(* IEC 61131-3 sources: CodigoPPC/Variaveis, 8 files *)

(* ---- GVL_Alarm.st ---- *)
{attribute 'qualified_only'}
VAR_GLOBAL
    // ─────────────────────────────────────────────────────────
    // ALARM MANAGER FLAGS (condições booleanas)
    // ─────────────────────────────────────────────────────────

	// Falhas na inicialização
    WARN_INV_CHECK_PARTIAL          : BOOL := FALSE;  // Inversores ausentes mas acima do limiar
	CRIT_SERIAL_INIT_FAIL			: BOOL := FALSE;	// Critico - Falha para iniciar as seriais
	CRIT_K1_TIMEOUT 				: BOOL := FALSE;    // Critico - falha na inicialização de K1 - falta detectar fechamento
	CRIT_K2_TIMEOUT 				: BOOL := FALSE;    // Critico - falha na inicialização de K2 - falta detectar fechamento
    CRIT_INV_CHECK_BELOW_THRESHOLD  : BOOL := FALSE;  // Respondentes < limiar → stError

    // Medição / Medidor
    ALARM_MEAS_MODBUS_TIMEOUT      	: BOOL := FALSE;  	// timeout de leitura (READ)
    ALARM_MEAS_MODBUS_ERRO       	: BOOL := FALSE;  	// xError do medidor (READ)
    ALARM_MEAS_FROZEN	            : BOOL := FALSE;  	// diagnosticCode = A900 (se aplicável)
    ALARM_MEAS_USING_LAST_VALUEU	: BOOL := FALSE;  	// bPoucosErros=TRUE e bDadosOK=FALSE
	ALARM_MEAS_RANGE_ERROR    		: BOOL := FALSE;    // Warning: Valor fora de faixa
    ALARM_MEAS_XCHECK_FAIL   		: BOOL := FALSE;    // Warning: Validação cruzada
    CRIT_MEAS_PERSISTENT_FAIL		: BOOL := FALSE;  	// bPoucosErros = FALSE
    CRIT_MEAS_MODBUS_TIMEOUT      	: BOOL := FALSE;  	// timeout de leitura (READ) repeticao fora da tolerancia
    CRIT_MEAS_MODBUS_ERRO       	: BOOL := FALSE;  	// xError do medidor (READ)  repeticao fora da tolerancia
	CRIT_MEAS_INIC_ERRO_TIMEOUT		: BOOL := FALSE;    // falha no teste de comunicação na inicialização do medidor

    // Comunicação inversores
    CRIT_COM_CHANNEL_FAIL           : BOOL := FALSE;  	// falha geral de comunicação → FAIL/STOP
	CRIT_CH1_MODBUS_TIMEOUT        	: BOOL := FALSE; 	// Canal COM1 TIMEOUT 3x
    CRIT_CH2_MODBUS_TIMEOUT        	: BOOL := FALSE; 	// Canal COM2 TIMEOUT 3x
	CRIT_CH1_MODBUS_ERRO	       	: BOOL := FALSE;  	// >50% falhas COM1 no ciclo
    CRIT_CH2_MODBUS_ERRO        	: BOOL := FALSE;  	// >50% falhas COM2 no ciclo

    // Sistema
	ALARM_SCAN_OVERRUN        		: BOOL := FALSE;    // Warning: Watchdog de ciclo
    CRIT_TC_POWER_NOT_SET           : BOOL := FALSE;    // TC_Power_kW = 0 na inicialização
    CRIT_NO_INVERTERS        		: BOOL := FALSE;    // Error: Nenhum inversor configurado
    CRIT_RTC_FAIL            		: BOOL := FALSE;    // Error: Falha RTC
    CRIT_INSTALLED_PWR_ZERO  		: BOOL := FALSE;    // Error: Potência instalada = 0
	CRIT_INSTALLED_SMAX_ZERO  		: BOOL := FALSE;    // Error: Potência reativa instalada = 0
	CRIT_SCAN_OVERRUN        		: BOOL := FALSE;    // CRITICO: Watchdog de ciclo 3x

    // Proteções normativas
    CRIT_HARDLIMIT_15S       		: BOOL := FALSE;    // Error: P > LPI+10% por >15s
    CRIT_EXPORT_OVER_LPI_30S   		: BOOL := FALSE;    // Error: P > LPI por >30s
    CRIT_K2_NOT_OPENED       		: BOOL := FALSE;    // Error: K2 não abriu após trip
	CRIT_MEAS_TIMEOUT_IN_FAIL    	: BOOL := FALSE;	// 5s sem medição válida em FAIL → STOP
	CRIT_FAIL_ENTRY                 : BOOL := FALSE;    // Entrada no estado FAIL

	// Status do sistema
	ALARM_FAIL_ACTIVE				: BOOL := FALSE;  	// MachineState=FAIL
    CRIT_STOP_ACTIVE	            : BOOL := FALSE;  	// MachineState=STOP
	CRIT_SCHEDULE_INDEX_INVALID		: BOOL := FALSE;    // Dia ou hora da semana inválido (CRITICAL)

    // ── Controle / PF ──
    ALARM_PF_BELOW_TARGET     		: BOOL := FALSE;    // Warning: PF < 0.92
    ALARM_PF_CRITICAL         		: BOOL := FALSE;    // Error: PF < 0.92 + Q saturado
    ALARM_Q_LIMITED_BY_SMAX    		: BOOL := FALSE;    // Info: Q limitado por S

	// FAIL-SAFE avançado
	ALARM_FAIL_RECOVERY_STARTED     : BOOL := FALSE;    // Timer de recuperação iniciou
	CRIT_FAIL_WRITE_FAILED          : BOOL := FALSE;    // Escrita zero falhou (inversores não responderam)
	CRIT_FAIL_WRITE_EXHAUSTED       : BOOL := FALSE;    // Esgotou retentativas de escrita zero → STOP
	CRIT_FAIL_GLOBAL_TIMEOUT        : BOOL := FALSE;    // Permaneceu em FAIL além do máximo permitido

	    // ── TURNOFF ──
    ALARM_TURNOFF_ACTIVE            : BOOL := FALSE;    // MachineState = TURNOFF
    CRIT_TURNOFF_WRITE_EXHAUSTED    : BOOL := FALSE;    // Escrita zero esgotou tentativas
    CRIT_TURNOFF_VERIFY_TIMEOUT     : BOOL := FALSE;    // Timeout verificação geração
    CRIT_TURNOFF_K2_NOT_OPENED      : BOOL := FALSE;    // K2 não abriu após trip controlado
	CRIT_TURNOFF_K1_NOT_OPENED      : BOOL := FALSE;    // K1 não abriu após comando

END_VAR

(* ---- GVL_ALARM_MANAGER.st ---- *)
{attribute 'qualified_only'}
VAR_GLOBAL
    // ─────────────────────────────────────────────────────────
    // ALARM MANAGER FLAGS (condições booleanas)
    // ─────────────────────────────────────────────────────────

	// Falhas na inicialização
	CRIT_SERIAL_INIT_FAIL			: BOOL := FALSE;	// Critico - Falha para iniciar as seriais
	CRIT_K1_TIMEOUT 				: BOOL := FALSE;    // Critico - falha na inicialização de K1 - falta detectar fechamento
	CRIT_K2_TIMEOUT 				: BOOL := FALSE;    // Critico - falha na inicialização de K2 - falta detectar fechamento

    // Medição / Medidor
    ALARM_MEAS_MODBUS_TIMEOUT      	: BOOL := FALSE;  	// timeout de leitura (READ)
    ALARM_MEAS_MODBUS_ERRO       	: BOOL := FALSE;  	// xError do medidor (READ)
    ALARM_MEAS_FROZEN	            : BOOL := FALSE;  	// diagnosticCode = A900 (se aplicável)
    ALARM_MEAS_USING_LAST_VALUEU	: BOOL := FALSE;  	// bPoucosErros=TRUE e bDadosOK=FALSE
	ALARM_MEAS_RANGE_ERROR    		: BOOL := FALSE;    // Warning: Valor fora de faixa
    ALARM_MEAS_XCHECK_FAIL   		: BOOL := FALSE;    // Warning: Validação cruzada
    CRIT_MEAS_PERSISTENT_FAIL		: BOOL := FALSE;  	// bPoucosErros = FALSE
    CRIT_MEAS_MODBUS_TIMEOUT      	: BOOL := FALSE;  	// timeout de leitura (READ) repeticao fora da tolerancia
    CRIT_MEAS_MODBUS_ERRO       	: BOOL := FALSE;  	// xError do medidor (READ)  repeticao fora da tolerancia

    // Comunicação inversores
    CRIT_COM_CHANNEL_FAIL           : BOOL := FALSE;  	// falha geral de comunicação → FAIL/STOP
	CRIT_CH1_MODBUS_TIMEOUT        	: BOOL := FALSE; 	// Canal COM1 TIMEOUT 3x
    CRIT_CH2_MODBUS_TIMEOUT        	: BOOL := FALSE; 	// Canal COM2 TIMEOUT 3x
	CRIT_CH1_MODBUS_ERRO	       	: BOOL := FALSE;  	// >50% falhas COM1 no ciclo
    CRIT_CH2_MODBUS_ERRO        	: BOOL := FALSE;  	// >50% falhas COM2 no ciclo

    // Sistema
	ALARM_SCAN_OVERRUN        		: BOOL := FALSE;    // Warning: Watchdog de ciclo
    CRIT_TC_POWER_NOT_SET           : BOOL := FALSE;    // TC_Power_kW = 0 na inicialização
    CRIT_NO_INVERTERS        		: BOOL := FALSE;    // Error: Nenhum inversor configurado
    CRIT_RTC_FAIL            		: BOOL := FALSE;    // Error: Falha RTC
    CRIT_INSTALLED_PWR_ZERO  		: BOOL := FALSE;    // Error: Potência instalada = 0
	CRIT_INSTALLED_SMAX_ZERO  		: BOOL := FALSE;    // Error: Potência reativa instalada = 0
	CRIT_SCAN_OVERRUN        		: BOOL := FALSE;    // CRITICO: Watchdog de ciclo 3x

    // Proteções normativas
    CRIT_HARDLIMIT_15S       		: BOOL := FALSE;    // Error: P > LPI+10% por >15s
    CRIT_EXPORT_OVER_LPI_30S   		: BOOL := FALSE;    // Error: P > LPI por >30s
    CRIT_K2_NOT_OPENED       		: BOOL := FALSE;    // Error: K2 não abriu após trip
	CRIT_MEAS_TIMEOUT_IN_FAIL    	: BOOL := FALSE;	// 5s sem medição válida em FAIL → STOP
	CRIT_FAIL_ENTRY                 : BOOL := FALSE;    // Entrada no estado FAIL

	// Status do sistema
	ALARM_FAIL_ACTIVE				: BOOL := FALSE;  	// MachineState=FAIL
    CRIT_STOP_ACTIVE	            : BOOL := FALSE;  	// MachineState=STOP
	CRIT_SCHEDULE_INDEX_INVALID		: BOOL := FALSE;    // Dia ou hora da semana inválido (CRITICAL)

    // ── Controle / PF ──
    ALARM_PF_BELOW_TARGET     		: BOOL := FALSE;    // Warning: PF < 0.92
    ALARM_PF_CRITICAL         		: BOOL := FALSE;    // Error: PF < 0.92 + Q saturado
    ALARM_Q_LIMITED_BY_SMAX    		: BOOL := FALSE;    // Info: Q limitado por S
END_VAR

(* ---- GVL_Comm.st ---- *)
{attribute 'qualified_only'}
(* ═══════════════════════════════════════════════════════════════════════
   GVL_Comm — Área de dados da comunicação Modbus RTU programática
   ═══════════════════════════════════════════════════════════════════════
   Esta GVL é o ponto de interface entre a Task_ModbusComm (que executa
   a comunicação) e a Task_Main (que executa o controle).

   Capacidade:
   COM1: 1 medidor + até 15 inversores
   COM2: até 15 inversores
   Canais de escrita por inversor: até 20 (índices 0..19)

   REGRA DE CONCORRÊNCIA (escritor único):
     - Task_ModbusComm ESCREVE: bCOMxConnected, bMeterOnline,
       bMeterReadDone, eMeterResult, awMeterRawData,
       bInvReadDone_COMx, eInvResult_COMx
     - Task_Main ESCREVE: bWritePendingCOMx, setpoints
     - Task_ModbusComm LÊ: bWritePendingCOMx, setpoints
   ═══════════════════════════════════════════════════════════════════════ *)
{attribute 'qualified_only'}

VAR_GLOBAL CONSTANT
    MAX_INV_PER_COM     	: UINT := 15;       // Inversores por porta COM
    MAX_WRITE_CHANNELS  	: UINT := 20;       // Canais de escrita por inversor (0..19)
END_VAR

VAR_GLOBAL
    // ─── Estado das portas COM ───────────────────────────────────
    bCOM1Connected      : BOOL;
    bCOM2Connected      : BOOL;
    bCOM1Error          : BOOL;
    bCOM2Error          : BOOL;

    // ─── Medidor (COM1) — Buffer raw para UN_chint/UN_URP1439 ───
    bMeterOnline        : BOOL;
    bMeterReadDone      : BOOL;
    eMeterResult        : E_ModbusResult;
    awMeterRawData      : ARRAY[0..63] OF WORD;
    uiMeterRegsRead     : UINT;

    // ─── Inversores COM1 — status de resposta ────────────────────
    abInvOnline_COM1        : ARRAY[1..15] OF BOOL;
    uiInvOnlineCount_COM1   : UINT;

    // ─── Inversores COM2 — status de resposta ────────────────────
    abInvOnline_COM2        : ARRAY[1..15] OF BOOL;
    uiInvOnlineCount_COM2   : UINT;

    // ─── Escrita — flags de pendência ────────────────────────────
    bWritePendingCOM1   : BOOL;
    bWritePendingCOM2   : BOOL;

    // ─── Configuração de slaves (preenchidos no stInit) ──────────
    uiMeterSlaveId      : UINT := 100;
    auiInvSlaveIdsCOM1  : ARRAY[1..15] OF UINT;
    auiInvSlaveIdsCOM2  : ARRAY[1..15] OF UINT;
    auiWriteRegAddr     : ARRAY[0..19] OF UINT;    // Endereço de registro por canal (0..19)

    // ─── Configuração geral ──────────────────────────────────────
    bConfigLoaded       : BOOL;
    bCommInitDone       : BOOL;
END_VAR

(* ---- GVL_Log.st ---- *)
{attribute 'qualified_only'}
// ════════════════════════════════════════════════════════════════════
// GVL_EventLog — Constantes do sistema de log de eventos
// ════════════════════════════════════════════════════════════════════
// Autor: Eng. Principal / Revisão Técnica PPC-GD
// Plataforma: WAGO CC100 (751-9402) / CODESYS V3.5 SP21 Patch 4
//
// DIMENSIONAMENTO:
//   64 entradas × 28 bytes = ~1.792 bytes de RETAIN
//   WAGO CC100 possui ~32 kB RETAIN → uso < 6%
//   Com ~1 evento/min, cobre >1 hora de histórico completo
//   Com taxa de pico (~10 eventos em cascata), ainda retém >6 min
// ════════════════════════════════════════════════════════════════════
{attribute 'qualified_only'}
VAR_GLOBAL CONSTANT
    MAX_EVENT_ENTRIES   : UINT := 64;   // Tamanho do ring buffer (potência de 2 facilita debug)
END_VAR

(* ---- GVL_Main.st ---- *)
{attribute 'qualified_only'}
VAR_GLOBAL CONSTANT

    // Parâmetros do sistema
    SOFTVERSION          		: UINT := 21;   					// Versão da aplicação
	DATAAPLICATION				: DATE := DATE#2025-12-05;			// Data da aplicação
	NMAXINVERSORES				: UINT := 30;						// Capacidade máxima de inversores
	TIPOSINVERSORES				: UINT := 8;						// total de inversores diferentes que podem estar presentes
	NDATASESPECIAIS 			: UINT := 48; 						// Quantidade de datas especiais disponíveis ao todo (para 10 anos)
	TIMEZONEOFFSET				: DINT := -3;
    CYCLE_TIME_MS				: UDINT := 1000;  					// tempo de ciclo de controle
	MAX_Meas_MODBUS_ERROS		: UDINT := 3;						// quantidade de erros permitido na leitura do medidor
	MAX_Meas_MODBUS_TIMEOUTS	: UDINT := 3;						// quantidade de timeouts permitido na leitura do medidor

END_VAR

VAR_GLOBAL
	timestampUTC				: UDINT;
	Result 						: RTS_IEC_RESULT;
  	ControlCycle    			: REAL:=1;            					// Tempo de ciclo de controle em SEGUNDOS (ex: 1.0 = 1 segundo)
	MachineState				: E_MachineState:= E_MachineState.START;
	fbEventLog 					: FB_EventLog;						// Function Block de registro de eventos

	CYCLE_TIME_TOLERANCE		: UDINT := 1200;  					// tolerancia de ultrapassagem para tempo de ciclo de controle de 20%

	// Saidas digitais
  	K1_out  					: BOOL;   							// DI X5_1 - K1 - controle permissivo
	K2_out						: BOOL;								// DI X5_2 - K2 - controle trip
  	LedRedOut					: BOOL;								// DI X5_3 - nada pronto - K1 e K2 abertos
  	LedYellowOut  				: BOOL;   							// DI X5_4 - K1 fechou - permissivo ok
  	LedGreenOut  				: BOOL;   							// DI X5_5 - K2 fechou - acende verde -tudo pronto

	// Entredas digitais
	K1_in        				: BOOL;                				// DI X12_1 - contato auxliar de K1_in=1 => K1 fechado (permite gerar)
  	K2_in        				: BOOL;                				// DI X12_2 - contato auxliar de K2_in=1 => K2 fechado (permite gerar) trip desarmado

    // Comandos da IHM
    // ─────────────────────────────────────────────────────────────
  	HMI_StartResetButton     	: BOOL := FALSE;           			// DI X12_3 - botao frontal para comandar ligar/reset geral quando no estado STOP
    HMI_TurnOffButton    		: BOOL := FALSE;  					// DI X12_4 "Desligar controlado"

    //    Medições (REAL) - Tensões (V), Correntes (A), Potências Ativas (W), Potências Reativas (var), PF (adimensional, sinal: + indutivo, - capacitivo)

    Ua  			: REAL := 0.0; // Tensão de fase A   - 2006H - Tensão de fase A em Volts (x 0,1 V)
    Ub  			: REAL := 0.0; // Tensão de fase B   - 2008H - Tensão de fase B em Volts (x 0,1 V)
    Uc  			: REAL := 0.0; // Tensão de fase C   - 200AH - Tensão de fase C em Volts (x 0,1 V)

	Ia    			: REAL 	:= 0.0; // 200CH - Corrente de fase A em A (x 0,001 A)
	Ib    			: REAL 	:= 0.0; // 200EH - Corrente de fase B em A (x 0,001 A)
	Ic    			: REAL 	:= 0.0; // 2010H - Corrente de fase C em A (x 0,001 A)

	Pt    			: REAL 	:= 0.0; // 2012H - Potencia ativa combinada em kW (x 0.1 para W, x 0.0001 para kW)
	Pa    			: REAL 	:= 0.0; // 2014H - Potencia ativa fase A 	em kW (x 0.1 para W, x 0.0001 para kW)
	Pb    			: REAL 	:= 0.0; // 2016H - Potencia ativa fase B 	em kW (x 0.1 para W, x 0.0001 para kW)
	Pc    			: REAL 	:= 0.0; // 2018H - Potencia ativa fase C    em kW (x 0.1 para W, x 0.0001 para kW)

	Qt    			: REAL 	:= 0.0; // 201AH - Potencia reativa combinada em kvar (x 0.1 para var, x 0.0001 para kvar)
	Qa    			: REAL 	:= 0.0; // 201CH - Potencia reativa fase A	 em kvar (x 0.1 para var, x 0.0001 para kvar)
	Qb    			: REAL 	:= 0.0; // 201EH - Potencia reativa fase B	 em kvar (x 0.1 para var, x 0.0001 para kvar)
	Qc    			: REAL 	:= 0.0; // 2020H - Potencia reativa fase C	 em kvar (x 0.1 para var, x 0.0001 para kvar)

	PFt    			: REAL 	:= 0.0; // 202AH - Fator de potência combinado (número positivo: indutivo, número negativo: capacitivo) (x0,001)
	PFa    			: REAL 	:= 0.0; // 202CH - Fator de potência de fase A (número positivo: indutivo, número negativo: capacitivo) (x0,001)
	PFb    			: REAL 	:= 0.0; // 202EH - Fator de potência de fase B (número positivo: indutivo, número negativo: capacitivo) (x0,001)
	PFc    			: REAL 	:= 0.0; // 2030H - Fator de potência de fase C (número positivo: indutivo, número negativo: capacitivo) (x0,001)

	// definição medidores dos dois canais de comunicação
	trigMedidor100  : BOOL;
	pMedidor100		: POINTER TO ModbusSlaveComPort;
	trigMedidor200  : BOOL;
	pMedidor200		: POINTER TO ModbusSlaveComPort;

	// definição dos inversores dos dois canais de comunicação
	MAX_CH1_MODBUS_ERROS		: UINT := 0;						// < 50% da quantidade de inversores sem ir para FAIL
	MAX_CH1_MODBUS_TIMEOUTS		: UINT := 0;						// < 50% da quantidade de inversores sem ir para FAIL
	MAX_CH2_MODBUS_ERROS		: UINT := 0;						// < 50% da quantidade de inversores sem ir para FAIL
	MAX_CH2_MODBUS_TIMEOUTS		: UINT := 0;						// < 50% da quantidade de inversores sem ir para FAIL
	trigInvCOM100				: ARRAY[1..15, 0..4] OF BOOL;
	trigInvCOM200				: ARRAY[1..15, 0..4] OF BOOL;
	NInversoresCOM01    		: UINT :=0;
	NInversoresCOM02    		: UINT :=0;
    pInversores100 	: ARRAY [1..15] OF POINTER TO ModbusSlaveComPort; 				// array de pointers para Inversor01..Inversor15 (apenas ponteiros - não recria instâncias)
	pInversores200 	: ARRAY [1..15] OF POINTER TO ModbusSlaveComPort; 				// array de pointers para Inversor01..Inversor15 (apenas ponteiros - não recria instâncias)

    //   COMANDOS E TELEMETRIA - Saídas do Controle

	// Potencia Total instalada e potencia Aparente Total instalada
  	InstalledPower 	: REAL; 														// Soma da potência nominal de todos os inversores ativos
	Q_max_permitido : REAL := 0.0;    												// Q máximo permitido (kvar)
	InstalledSmax   : REAL; 														// NOVO: Potência Aparente Máxima Total (kVA)

	// COMANDOS DE CONTROLE
	MaxExportLimit 	: REAL;              											// Limite de exportação do scheduler (kW)
	P_cmd_total_kW 	: REAL;              											// Comando total de P (kW)
	Q_cmd_total_kvar: REAL;            												// Comando total de Q (kvar)

    // Telemetria: Setpoint atual da agenda (antes das proteções)
    TotalPowerPercent : REAL;

    // Telemetria: Potência Reativa total desejada (kVA)
    TotalReactivePower : REAL;

    // Telemetria: Valores efetivos calculados para cada inversor
    P_inv_kW     	: ARRAY[1..NMAXINVERSORES] OF REAL; 							// valor de setpoint de potencia ativa em kW
	P_inv_Percent 	: ARRAY[1..NMAXINVERSORES] OF REAL; 							// valor de setpoint de potencia ativa em percentual do nominal
	P_inv_limit 	: ARRAY[1..NMAXINVERSORES] OF REAL; 							// valor limite de potencia ativa com base na SMAX de cada um
    Q_inv_kvar    	: ARRAY[1..NMAXINVERSORES] OF REAL; 							// valor de setpoint de potencia reativa em kVA
    PF_inv 			: ARRAY[1..NMAXINVERSORES] OF REAL; 							// valor do fator de potencia de cada inversor (deve ser 0,92 para todos)
	PF_inv_Percent	: ARRAY[1..NMAXINVERSORES] OF REAL; 							// valor de setpoint de fator de potencia em percentual

	// Margem de segurança para compensar erro de TC perto de zero, o sistema tentará manter importação mínima garantido que não haja exportação
	SafetyMargin_pct: REAL :=0.03;
	TC_Power_kW		: REAL := 0.0; // deve ser configurado como 3% da potencia total sob controle pelo TC

	// ════════════════════════════════════════════════════════════════
	// DIAGNÓSTICO DE PF
	// ════════════════════════════════════════════════════════════════
	Q_available_max : REAL;             											// Q máximo disponível (kvar)
	PF_effective 	: REAL;                											// PF efetivo resultante
	PFErro 			: BOOL;                   										// TRUE = PF < 0.92 não atingível (banco de capacitores)

	// ════════════════════════════════════════════════════════════════
    // DIAGNÓSTICO DE FATOR DE POTÊNCIA
    // ════════════════════════════════════════════════════════════════

    // Status geral
    PF_target : REAL := 0.92;                   // PF alvo (mínimo aceitável)
    PF_measured : REAL;                         // PF medido no ponto de conexão
    PF_achieved : REAL;                         // PF efetivamente alcançado após compensação
    PF_OK : BOOL;                               // TRUE = PF ≥ 0.92

    // Potências
    P_generated_kW : REAL;                      // P total gerado pelos inversores
    P_allocated_kW : REAL;                      // P efetivamente alocado
    Q_measured_kvar : REAL;                     // Q medido no ponto de conexão (carga)
    Q_required_kvar : REAL;                     // Q necessário para atingir PF ≥ 0.92
    Q_commanded_kvar : REAL;                    // Q comandado pelo FB_PIQ
    Q_available_kvar : REAL;                    // Q que inversores conseguem fornecer
    Q_allocated_kvar : REAL;                    // Q efetivamente alocado
    Q_deficit_kvar : REAL;                      // Déficit de Q (se > 0, falta Q)

    // Capacidade dos inversores
    S_total_available_kVA : REAL;               // S total disponível (soma de todos inversores)
    S_total_used_kVA : REAL;                    // S total utilizado
    S_utilization_pct : REAL;                   // % de utilização de S
    Q_capacity_total_kvar : REAL;               // Capacidade total de Q dos inversores (atual)
    Q_utilization_pct : REAL;                   // % de utilização de Q

    // Diagnóstico e recomendações
    Q_deficit_percent : REAL;                   // Déficit de Q em % do necessário
    Capacitor_bank_size_kvar : REAL;            // Tamanho recomendado de banco de capacitores
    Capacitor_bank_recommended : BOOL;          // TRUE = Recomenda banco de capacitores
    PF_alarm_code : UINT;                       // Código de alarme (0=OK, 1=Aviso, 2=Crítico)

    // Histórico (opcional)
    PF_min_24h : REAL := 1.0;                   // PF mínimo nas últimas 24h
    PF_avg_24h : REAL := 1.0;                   // PF médio nas últimas 24h
    Q_deficit_max_24h : REAL;                   // Déficit máximo de Q nas últimas 24h
    PF_alarm_count_24h : UDINT;                 // Quantidade de alarmes nas últimas 24h

    // Inversores individuais (diagnóstico detalhado)
    Inv_S_utilization : ARRAY[1..NMAXINVERSORES] OF REAL;  // % S usado por inversor
    Inv_Q_available : ARRAY[1..NMAXINVERSORES] OF REAL;    // Q disponível por inversor (kvar)
    Inv_limited : ARRAY[1..NMAXINVERSORES] OF BOOL;        // TRUE = Inversor limitado por S
END_VAR

(* ---- GVL_ModbusProfiles.st ---- *)
(* ═══════════════════════════════════════════════════════════════════════
   GVL_ModbusProfiles — Perfis de dispositivos Modbus
   ═══════════════════════════════════════════════════════════════════════
   Contém os perfis hardcoded de cada modelo de inversor suportado.
   Declarados como CONSTANT: imutáveis em runtime, residem em Flash.

   FASE 1: apenas Goodwe GW50K-MT (único modelo em operação).
   FASE 4: FB_LoadProfiles substituirá estes valores por dados do CSV,
           mantendo este como fallback em caso de falha de leitura.

   PROTOCOLO GOODWE — REGISTRO 0x0101 (Fator de Potência):
     Indutivo  (Q ≥ 0): valor 80..100 → PF = valor / 100  (ex: 92 → PF 0.92)
     Capacitivo(Q < 0): valor  1.. 20 → PF = (100-valor)/100 (ex: 10 → PF 0.90 cap)
     A conversão para este formato já é feita pelo FB_QAlloc e armazenada
     em GVL_Main.PF_inv_Percent[i]. Aqui Scale=1.0 pois o valor já está
     no formato correto para o registro.

   PROTOCOLO GOODWE — REGISTRO 0x0100 (Potência Ativa):
     Valor direto 0..100 representando 0..100% da potência nominal.
     FB_PAlloc já calcula P_inv_Percent em 0..100. Scale=1.0.
   ═══════════════════════════════════════════════════════════════════════ *)
{attribute 'qualified_only'}
VAR_GLOBAL CONSTANT

    Profile_Goodwe_GW50K : ST_InverterProfile := (
        Name             := 'Goodwe GW50K-MT',
        ManufacturerCode := 1,          // 1 = Goodwe
        MaxRegsPerWrite  := 1,          // Goodwe: 1 registro por transação FC06
        InterFrameDelayMs := 0,         // ModbusFB respeita silêncio RTU automaticamente

        nWriteRegs := 2,
        WriteMap := [
            // Índice 0 — Setpoint Potência Ativa (%)
            (Address     := 16#0100,    // 256 decimal
             Quantity    := 1,
             FuncCode    := 6,          // FC06: Write Single Register
             Scale       := 1.0,        // P_inv_Percent já está em 0..100
             Offset      := 0.0,
             MinPhys     := 0.0,        // 0% = inversor parado
             MaxPhys     := 100.0,      // 100% = potência nominal
             bEnabled    := TRUE),

            // Índice 1 — Setpoint Fator de Potência (formato Modbus Goodwe)
            // Indutivo:  80..100 (PF = valor/100)
            // Capacitivo: 1..20  (PF = (100-valor)/100)
            // PF_inv_Percent já contém o valor neste formato (calculado em FB_QAlloc)
            (Address     := 16#0101,    // 257 decimal
             Quantity    := 1,
             FuncCode    := 6,          // FC06: Write Single Register
             Scale       := 1.0,        // PF_inv_Percent já é o valor de registro
             Offset      := 0.0,
             MinPhys     := 1.0,        // menor valor válido do protocolo
             MaxPhys     := 100.0,      // maior valor válido (PF=1.0 indutivo)
             bEnabled    := TRUE),

            // Índices 2..4 — reservados
            (bEnabled := FALSE, Scale := 1.0, MinPhys := 0.0, MaxPhys := 0.0,
             Address := 0, Quantity := 0, FuncCode := 0, Offset := 0.0),
            (bEnabled := FALSE, Scale := 1.0, MinPhys := 0.0, MaxPhys := 0.0,
             Address := 0, Quantity := 0, FuncCode := 0, Offset := 0.0),
            (bEnabled := FALSE, Scale := 1.0, MinPhys := 0.0, MaxPhys := 0.0,
             Address := 0, Quantity := 0, FuncCode := 0, Offset := 0.0)
        ]
    );

END_VAR

(* ---- GVL_Pers.st ---- *)
{attribute 'qualified_only'}
VAR_GLOBAL PERSISTENT RETAIN

    // CONFIGURAÇÕES DO SISTEMA (Dados que não podem ser perdidos no desligamento)

	// Definição do medidor a ser usado
	MeasDeviceType 		: E_MeasDeviceType := E_MeasDeviceType.CHINT_DTSU666;
	RTC					: UINT;													// razão de transformação do TC
	RTP					: UINT;													// razão de transformação do TP

    // Potência nominal (kW) por tipo
    InvActivePower 		: ARRAY[1..GVL_Main.NMAXINVERSORES] OF REAL; 		// kW
    // Potência Aparente Máxima (kVA) por tipo
    InvSmaxPower 		: ARRAY[1..GVL_Main.NMAXINVERSORES] OF REAL;		// kVA

    // --- Parâmetros de Controle de Exportação ---
    PowerMode 			: UINT := 2;      								// 0=Total, 1=Por Fase, 2=Ambos
	OperationMode		: BOOL := TRUE;									// FALSE=Export Control  TRUE=Zero Grid
	ControlMode			: UINT := 1;									// 0 = manual  1 = automatico (PI ativo)
    TotALARMaxExport_kW : REAL := 0; 									// Limite físico total (kW)
    PhaseMaxExport_kW 	: REAL := 0; 									// Limite físico por fase (kW)

	// Definição do numero de canais em COM1 e COM2
	nChannelsToWriteCOM1	 	: UINT :=2;
	nChannelsToWriteCOM2	 	: UINT :=2;

    (*
	Regra prática para GD solar: Ti entre 5s e 20s. Mais rápido pode oscilar com a latência Modbus.
	Mais lento perde capacidade de compensar nuvens passando.
	Ti é o Tempo Integral do controlador PI, também chamado de tempo de reset.
	Relação Ki= Kp / Ti   Então se você tem Kp = 1.0 e Ti = 10s => Ki=1.0/10 = 0.1 (por segundo)
	Na prática para seu sistema:
	Ti pequeno (ex: 2s) → integral age rápido → mais agressivo → risco de oscilação
	Ti grande (ex: 30s) → integral age devagar → mais conservador → lento para corrigir erro estacionário
	Ti = 10s → o controlador elimina o erro estacionário em aproximadamente 30 a 40 segundos (≈ 3-4 × Ti)
	Resumo em uma frase:
	Ti = 10s é "quanto tempo o integrador leva para alcançar a mesma força que o proporcional já deu instantaneamente".
	*)

	// --- Controle Droop (Potência Ativa) ---
	Droop_Enable     	: BOOL := TRUE;      							// Habilita droop
	K_Droop          	: REAL := 0.15;      							// kW/kW  (ex.: 0.05 = 5% de ganho)
	Deadband_Droop   	: REAL := 2.0;       							// % (erro menor não gera droop)
	Droop_Max        	: REAL := 0.4;       							// Fração da potência instalada (ex.: 0.6 = 60%)

	// --- Parâmetros do Controlador PI (Potência Ativa) ---
    Kp_P           		: REAL := 0.25;									// Recomendado: 0.1 a 1.0
																	    // Maior → resposta mais rápida, risco de oscilação
																	    // Menor → mais suave, mas mais lento
    Ki_P           		: REAL := 0.02;									// Recomendado: 0.02 a 0.1 - Com 1s de ciclo e tempo morto ~1,2–1,6s, integral muito alto oscila.
																		// Com T=1s: constante de tempo integral Ti = Kp/Ki = 12,5s
																	    // Significado: elimina erro estacionário em ~10 segundos
																	    // NUNCA > 0.2 com T=1s (oscilação garantida)
	RampUp_P 			: REAL := 15.0;           						// Rampa de subida (kW/s) - limitar a 15-20 kW/s por causa do sweep de setpoints nos inversores
	RampDown_P 			: REAL := 20.0;         						// Rampa de descida (kW/s) - RampDown_P ≤ 20–30 kW/s
    Deadband_P  		: REAL := 1.0;  								// % da potência instalada (ex: 1.0 = 1%)

    // --- Configuração de Fator de Potência (PF) e Reativos (Q) ---
    PF_target       	: REAL := 0.92; 								// Alvo |PF|
	PF_sign				: REAL := 1.0;

    // Parâmetros do PI de Correção de Q (Feedforward + Feedback)
    Kp_Q           		: REAL := 50.0;									// Recomendado: 20.0 a 100.0 kvar/pu_PF
																	    // Unidade: kvar por unidade de erro de PF
																	    // Ex: erro PF = 0.02 → P_term = 50 * 0.02 = 1.0 kvar
    Ki_Q           		: REAL := 5.0;									// Recomendado: 2.0 a 10.0 kvar/(pu_PF·s
																	    // Com T=1s: Ti = Kp/Ki = 10s => elimina erro em ~30-40s
																	    // Significado: corrige PF em ~10 segundos
	RampUp_Q 			: REAL := 50.0;            						// Rampa de subida (kvar/s)
	RampDown_Q 			: REAL := 50.0;          						// Rampa de descida (kvar/s)
	Deadband_Q 			: REAL := 0.01;          						// Zona morta de PF (ex: 0.01 = ±0.01) — padrão para GD

    // --- Histerese de Habilitação ---
    HysteresisOn	   	: REAL := 0.01; 								// Liga controle acima de 1%
    HysteresisOff		: REAL := 0.01; 								// Desliga abaixo de 1%

    // --- Agenda Semanal (7 dias x 24 horas) e Datas Especiais
	bHorarioVerao 		: BOOL:= FALSE;									// se TRUE  = Horário de Verão Ativo (+1h)
    WeekSchedule_kW 	: ARRAY[1..7, 1..24] OF REAL; 					// (1=Dom 2=Seg 3=Ter 4=Quarta 5=Quinta 6=Sexta 7=Sábado) em kW
    DatasEspeciais   	: ARRAY[1..GVL_Main.NDATASESPECIAIS] OF DATE;		// inicializa com zeros
	SpecialDaySchedule 	: ARRAY[1..GVL_Main.NDATASESPECIAIS] OF REAL;		// cada data especial tem apenas um valor de potencia maxima valido para o dia inteiro

    // ════════════════════════════════════════════════════════════════
    // LIMITES FÍSICOS DO SISTEMA (Baseados no Transformador e Rede)
    // ════════════════════════════════════════════════════════════════
	// SafetyMargin_kW = SafetyMargin_pct × TC_Power_kW / 100 - Margem de segurança para compensar erro de TC perto de zero
	SafetyMargin_pct 	: REAL := 3.0;     								// Percentual do TC (%)
	// Exemplo 1: TC de 500 A, Tensão 380 V => P_TC = √3 × V × I = 1.732 × 380 × 500 = 329 kW
	TC_Power_kW			: REAL := 0.0; 									// deve ser configurado como 3% da potencia total sob controle pelo TC

	VMIN 				: REAL := 7170;  // Volts - tensão de fase minima para tensão primária de 13,8kV
    VMAX 				: REAL := 8370;  // Volts - tensão de fase máxima para tensão primária de 13,8kV
    IMAX 				: REAL := 125.0;  // Amperes - corrente de linha - para potencia de usina de 3MW erro transformador 5%
    PMAX 				: REAL := 3200.0; // kW (Demanda contratada + 10% de margem)
	QMAX				: REAL := 2400.0; // kvar tan(acos(0.8)) × Pmax
	// τ = tempo para atingir ~63% do valor final e T_scan = período de amostragem (1s no seu caso)
	// α = T_scan / (τ + T_scan)  => Alpha=0.5 => 3 segundos para atingir 95% do valor final
	// Item 2.1: "Responder em até 15 segundos a rejeição de carga"
	// Item 2.2: "Limitar exportação em até 15 segundos"
	// Nuvens passageiras: variação em 1–5 segundos
	// Rejeição de carga: instantânea (< 1s)
	// Ruído de medição: < 100 ms
	ALPHA				: REAL := 0.25;

END_VAR

(* ---- GVL_Persis.st ---- *)
{attribute 'qualified_only'}
VAR_GLOBAL PERSISTENT RETAIN

    // CONFIGURAÇÕES DO SISTEMA (Dados que não podem ser perdidos no desligamento)

	// Definição do medidor a ser usado
	MeasDeviceType 		: E_MeasDeviceType := E_MeasDeviceType.CHINT_DTSU666;

    // Potência nominal (kW) por tipo
    InvActivePower 		: ARRAY[1..GVL_Main.NMAXINVERSORES] OF REAL; 		// kW
    // Potência Aparente Máxima (kVA) por tipo
    InvSmaxPower 		: ARRAY[1..GVL_Main.NMAXINVERSORES] OF REAL;		// kVA

    // --- Parâmetros de Controle de Exportação ---
    PowerMode 			: UINT := 2;      								// 0=Total, 1=Por Fase, 2=Ambos
	OperationMode		: BOOL := TRUE;									// FALSE=Export Control  TRUE=Zero Grid
	ControlMode			: UINT := 1;									// 0 = manual  1 = automatico (PI ativo)
    TotALARMaxExport_kW : REAL := 0; 									// Limite físico total (kW)
    PhaseMaxExport_kW 	: REAL := 0; 									// Limite físico por fase (kW)

    (*
	Regra prática para GD solar: Ti entre 5s e 20s. Mais rápido pode oscilar com a latência Modbus.
	Mais lento perde capacidade de compensar nuvens passando.
	Ti é o Tempo Integral do controlador PI, também chamado de tempo de reset.
	Relação Ki= Kp / Ti   Então se você tem Kp = 1.0 e Ti = 10s => Ki=1.0/10 = 0.1 (por segundo)
	Na prática para seu sistema:
	Ti pequeno (ex: 2s) → integral age rápido → mais agressivo → risco de oscilação
	Ti grande (ex: 30s) → integral age devagar → mais conservador → lento para corrigir erro estacionário
	Ti = 10s → o controlador elimina o erro estacionário em aproximadamente 30 a 40 segundos (≈ 3-4 × Ti)
	Resumo em uma frase:
	Ti = 10s é "quanto tempo o integrador leva para alcançar a mesma força que o proporcional já deu instantaneamente".
	*)

	// --- Controle Droop (Potência Ativa) ---
	Droop_Enable     	: BOOL := TRUE;      							// Habilita droop
	K_Droop          	: REAL := 0.15;      							// kW/kW  (ex.: 0.05 = 5% de ganho)
	Deadband_Droop   	: REAL := 2.0;       							// % (erro menor não gera droop)
	Droop_Max        	: REAL := 0.4;       							// Fração da potência instalada (ex.: 0.6 = 60%)

	// --- Parâmetros do Controlador PI (Potência Ativa) ---
    Kp_P           		: REAL := 0.25;									// Recomendado: 0.1 a 1.0
																	    // Maior → resposta mais rápida, risco de oscilação
																	    // Menor → mais suave, mas mais lento
    Ki_P           		: REAL := 0.02;									// Recomendado: 0.02 a 0.1 - Com 1s de ciclo e tempo morto ~1,2–1,6s, integral muito alto oscila.
																		// Com T=1s: constante de tempo integral Ti = Kp/Ki = 12,5s
																	    // Significado: elimina erro estacionário em ~10 segundos
																	    // NUNCA > 0.2 com T=1s (oscilação garantida)
	RampUp_P 			: REAL := 15.0;           						// Rampa de subida (kW/s) - limitar a 15-20 kW/s por causa do sweep de setpoints nos inversores
	RampDown_P 			: REAL := 20.0;         						// Rampa de descida (kW/s) - RampDown_P ≤ 20–30 kW/s
    Deadband_P  		: REAL := 1.0;  								// % da potência instalada (ex: 1.0 = 1%)

    // --- Configuração de Fator de Potência (PF) e Reativos (Q) ---
    PF_target       	: REAL := 0.92; 								// Alvo |PF|
	PF_sign				: REAL := 1.0;
    // Parâmetros do PI de Correção de Q (Feedforward + Feedback)
    Kp_Q           		: REAL := 50.0;									// Recomendado: 20.0 a 100.0 kvar/pu_PF
																	    // Unidade: kvar por unidade de erro de PF
																	    // Ex: erro PF = 0.02 → P_term = 50 * 0.02 = 1.0 kvar
    Ki_Q           		: REAL := 5.0;									// Recomendado: 2.0 a 10.0 kvar/(pu_PF·s
																	    // Com T=1s: Ti = Kp/Ki = 10s => elimina erro em ~30-40s
																	    // Significado: corrige PF em ~10 segundos
	RampUp_Q 			: REAL := 50.0;            						// Rampa de subida (kvar/s)
	RampDown_Q 			: REAL := 50.0;          						// Rampa de descida (kvar/s)
	Deadband_Q 			: REAL := 0.01;          						// Zona morta de PF (ex: 0.01 = ±0.01) — padrão para GD

    // --- Histerese de Habilitação ---
    HysteresisOn	   	: REAL := 0.01; 								// Liga controle acima de 1%
    HysteresisOff		: REAL := 0.01; 								// Desliga abaixo de 1%

    // --- Agenda Semanal (7 dias x 24 horas) e Datas Especiais
	bHorarioVerao 		: BOOL:= FALSE;									// se TRUE  = Horário de Verão Ativo (+1h)
    WeekSchedule_kW 	: ARRAY[1..7, 1..24] OF REAL; 					// (1=Dom 2=Seg 3=Ter 4=Quarta 5=Quinta 6=Sexta 7=Sábado) em kW
    DatasEspeciais   	: ARRAY[1..GVL_Main.NDATASESPECIAIS] OF DATE;		// inicializa com zeros
	SpecialDaySchedule 	: ARRAY[1..GVL_Main.NDATASESPECIAIS] OF REAL;		// cada data especial tem apenas um valor de potencia maxima valido para o dia inteiro

    // ════════════════════════════════════════════════════════════════
    // LIMITES FÍSICOS DO SISTEMA (Baseados no Transformador e Rede)
    // ════════════════════════════════════════════════════════════════
	// SafetyMargin_kW = SafetyMargin_pct × TC_Power_kW / 100 - Margem de segurança para compensar erro de TC perto de zero
	SafetyMargin_pct 	: REAL := 3.0;     								// Percentual do TC (%)
	// Exemplo 1: TC de 500 A, Tensão 380 V => P_TC = √3 × V × I = 1.732 × 380 × 500 = 329 kW
	TC_Power_kW			: REAL := 0.0; 									// deve ser configurado como 3% da potencia total sob controle pelo TC

	VMIN 				: REAL := 7170;  // Volts - tensão de fase minima para tensão primária de 13,8kV
    VMAX 				: REAL := 8370;  // Volts - tensão de fase máxima para tensão primária de 13,8kV
    IMAX 				: REAL := 125.0;  // Amperes - corrente de linha - para potencia de usina de 3MW erro transformador 5%
    PMAX 				: REAL := 3200.0; // kW (Demanda contratada + 10% de margem)
	QMAX				: REAL := 2400.0; // kvar tan(acos(0.8)) × Pmax
	// τ = tempo para atingir ~63% do valor final e T_scan = período de amostragem (1s no seu caso)
	// α = T_scan / (τ + T_scan)  => Alpha=0.5 => 3 segundos para atingir 95% do valor final
	// Item 2.1: "Responder em até 15 segundos a rejeição de carga"
	// Item 2.2: "Limitar exportação em até 15 segundos"
	// Nuvens passageiras: variação em 1–5 segundos
	// Rejeição de carga: instantânea (< 1s)
	// Ruído de medição: < 100 ms
	ALPHA				: REAL := 0.25;

END_VAR
